(* FB Arbiter

The arbiter primary objectives are:
- Provide a simple interface for devices to request beam parameter sets
- Provide a way for devices to verify their BPS is active in the arbiter
- Provide a way for devices remove their requests from evaluation
- Evaluate all active beam parameter requests registered with the aribiter,
to determine the safest combination of all sets, provide this set as an output.
- Do all of this with minimal overhead

To these ends, the arbiter uses a hash-table, the rows being a state-id as the key, and a corresponding
 beam parameter set to be evaluated against all the other sets (or rows), in the table.
 
The hash table can be thought of as an array on steriods, they are worth reading about, suffice to say
the hash table will tell you when you reach the end of all the entries, and enables us to find entries quickly.

These features efficiently address the addition, removal, and verification of beam parameter sets listed in the above requirements.

An important thing to pay attention to is the A_Arbitrate action. This action implements the evaluation of beam parameter
sets against each other.

*)

FUNCTION_BLOCK FB_Arbiter
VAR_INPUT
	i_nStateID	:	UDINT; //Set to the stateID of the state requesting the beam parameter set
	i_stAssertBeamParams	:	ST_BeamParams; //Set to the beam parameter set of the state required
END_VAR
VAR_OUTPUT
	q_stBeamParams	:	ST_BeamParams; //Updated on each cycle of the arbiter FB with the current arbitrated beam parameter set
	
	q_xStateIDFound	:	BOOL; //Set true if a state-id is found in the assertion pool after calling A_VerifyAssertion
END_VAR
VAR
	
	fbBPAssertionPool	:	FB_BeamParamAssertionPool; //Table of active beam parameter assertions
	
	getPosPtr	: POINTER TO T_HashTableEntry := 0; 
	getBPStruct	:	ST_BeamParams;
	stOutputBP	:	ST_BeamParams; //Safest beam parameters from all in the assertion pool
	
	
END_VAR

//Arbitrate
(*
This step cycles through every hash table entry, comparing
the beam parameters from each assertion to what we're planning
to assert.

The safer of the two parameters is kept so at the end we may
have a mix of beam parameters, the composition being safe for
all asserters.

*)

//Safest parameters to start
stOutputBP := F_SetBeamParams(
	fAtt := 100,
	fPP_mJ := 0,
	fLower_eV := 0,
	fUpper_eV := 1800,
	nRate := 0
	);

fbBPAssertionPool.A_GetFirst( putPosPtr := 0, getPosPtr=>getPosPtr, getValue=>getBPStruct );
IF fbBPAssertionPool.bOk THEN
	
	//The first entry in the hash table is taken as the setting to arbitrate against
	stOutputBP := F_SetBeamParams(
		fAtt := getBPStruct.fAtt,
		fPP_mJ := getBPStruct.fPP_mJ,
		fLower_eV := getBPStruct.fLower_eV,
		fUpper_eV := getBPStruct.fUpper_eV,
		nRate := getBPStruct.nRate
	);

	REPEAT
		fbBPAssertionPool.A_GetNext( putPosPtr := fbBPAssertionPool.getPosPtr , getPosPtr=>getPosPtr, getValue=>getBPStruct );
		IF fbBPAssertionPool.bOk THEN
			A_Arbitrate();
		END_IF
	UNTIL NOT fbBPAssertionPool.bOk
	END_REPEAT

END_IF

q_stBeamParams := stOutputBP;

ACTION A_Arbitrate:

//Attenuation
//Add something here to register the key that won for each param
stOutputBP.fAtt := MAX(stOutputBP.fAtt, getBPStruct.fAtt);

//Pulse energy
stOutputBP.fPP_mJ := MIN(stOutputBP.fPP_mJ, getBPStruct.fPP_mJ);

//Photon energy ranges
stOutputBP.neVReqRange := stOutputBP.neVReqRange AND getBPStruct.neVReqRange;

//Rate
stOutputBP.nRate := MIN(stOutputBP.nRate, getBPStruct.nRate);
END_ACTION

ACTION A_AssertBP:
//fbTable.A_Add( key := 12345, putValue := putValue, getPosPtr=>getPosPtr, getValue=>getValue );

(* This action adds a state-id and beam parameter set to the beam parameter assertion pool (arbiter
hash table). Use like so:

fbArbiter.A_AssertBP(
i_nStateID := nStateID,
i_stAssertBeamParams := stDesiredBeamParams
);

*)

IF i_nStateID <> EXCLUDED_ASSERTION_ID THEN

	fbBPAssertionPool.A_Add(
		key := i_nStateID,
		putValue := i_stAssertBeamParams,
		getPosPtr=>getPosPtr,
		getValue => getBPStruct
	);
END_IF
	
IF NOT fbBPAssertionPool.bOk THEN
	; //Overflow <TODO>
END_IF
END_ACTION

ACTION A_Init:
// Clears the entire beam parameter assertion pool (hashtable).

fbBPAssertionPool.A_Reset();
END_ACTION

ACTION A_RemoveAssertion:

(* Searches for a state-id, and removes it from the assertion pool.

Use like so:
fbArbiter.A_RemoveAssertion(
i_nStateId := nStateIDAssertionToRemove
);

*)

IF i_nStateId <> EXCLUDED_ASSERTION_ID THEN
	fbBPAssertionPool.A_Remove(key := i_nStateId, getPosPtr=>getPosPtr, getValue=>getBPStruct);
	
	IF fbBPAssertionPool.bOk THEN
		;
	ELSE
		;
	END_IF
END_IF
END_ACTION

ACTION A_VerifyAssertion:

(* Searches state assertion pool for a state-id, and sets q_xStateIDFound true if found.

Use like so:

fbArbiter.A_VerifyAssertion(
i_nStateId := nStateIDAssertionToCheck
);

IF fbArbiter.q_xStateIDFound THEN:
	Do something
ELSE:
	Don't do something

*)

IF i_nStateID <> EXCLUDED_ASSERTION_ID THEN
	
	fbBPAssertionPool.A_Lookup( key := i_nStateID, getPosPtr=>getPosPtr, getValue=>getBPStruct );

	q_xStateIDFound	:= fbBPAssertionPool.bOk;

ELSE
	q_xStateIDFound := FALSE;
END_IF
END_ACTION

END_FUNCTION_BLOCK

(* stored: Version 1.1.0.1, ProductVersion 3.1.4022.12
   POU FB_Arbiter: Id {9cc1f6b7-c43c-0fbb-09be-271b21ce1be7}, SpecialFunc None
   Action A_Arbitrate: Id {cd232571-a3df-0041-3bcc-1fe44a9b9a88}
   Action A_AssertBP: Id {f6e89361-055c-0560-0933-bcdd7d87f7bb}
   Action A_Init: Id {31a8de0d-caf8-01fc-1b86-c0ff1708d44b}
   Action A_RemoveAssertion: Id {024321c3-bc6f-0692-0562-0a65dc09776d}
   Action A_VerifyAssertion: Id {905e28be-7804-0837-3111-bddd3e35d311} *)
